// TIA Portal V15.1 export
// export: Created 2024-05-17T05:38:38.7642875Z, ExportSetting WithDefaults, DisplayName Totally Integrated Automation Portal, DisplayVersion V15.1 Update 5, DisplayName TIA Portal Openness, DisplayVersion V15.1 Update 5, DisplayName SINAMICS Startdrive Advanced, DisplayVersion V15.1, DisplayName G130, G150, S120, S150, SINAMICS MV, S210, DisplayVersion V15.1, DisplayName G110M, G120, G120C, G120D, G120P, DisplayVersion V15.1, DisplayName STEP 7 Professional, DisplayVersion V15.1 Update 5, DisplayName STEP 7 Safety, DisplayVersion V15.1, DisplayName WinCC Professional, DisplayVersion V15.1 Update 5, DisplayName SIMATIC Visualization Architect, DisplayVersion V15.1
FUNCTION_BLOCK "LGBAndonHCall"   // FB6687, FBD
TITLE = LGBAndonHCall
{ S7_Optimized_Access := 'TRUE' }
VERSION : 0.1
// This module will evaluate if an Andon HCall from pullcords and/or buttons is 
// valid and make the Hcall(AndonLight) active. It sends the result to LAndonxMConfig
// stored: AutoNumber false, IsIECCheckEnabled false, IsRetainMemResEnabled false, MemoryReserve 100, SetENOAutomatically False, UDAEnableTagReadback false
   VAR_INPUT
      I_HCall { ExternalAccessible := 'False'; ExternalVisible := 'False'; ExternalWritable := 'False'} : Bool;   // Input of the Human Call
      I_PartPresent { ExternalAccessible := 'False'; ExternalVisible := 'False'; ExternalWritable := 'False'} : Bool;   // Part is present on workstation
      C_HCallNumber { ExternalAccessible := 'False'; ExternalVisible := 'False'; ExternalWritable := 'False'} : Int;   // Address of the human call 1-32
      C_WorkStationNumber { ExternalAccessible := 'False'; ExternalVisible := 'False'; ExternalWritable := 'False'} : Int;   // Addeess of the Andon Station
   END_VAR
   VAR_OUTPUT
      O_AndonActiveSignal { ExternalAccessible := 'False'; ExternalVisible := 'False'; ExternalWritable := 'False'} : Bool;   // Output of the Hcall Light
      O_AndonCycleStpAfter { ExternalAccessible := 'False'; ExternalVisible := 'False'; ExternalWritable := 'False'} : Bool;   // Stop after end of cycle
   END_VAR
   VAR_IN_OUT
      IO_AndonDataExchange : "AndonDataExchangeVCG";   // Andon dataExchange
      H_HMI : "H_HMI";   // Animation
      H_GBAndonHCal : "H_GBAndonHCall";   // Animation
   END_VAR
   VAR RETAIN
      AndonActiveSignal { ExternalAccessible := 'False'; ExternalVisible := 'False'; ExternalWritable := 'False'} : Bool;
   END_VAR
   VAR
      AndonHCallDW { ExternalAccessible := 'False'; ExternalVisible := 'False'; ExternalWritable := 'False'} : DWord;
   END_VAR
   VAR RETAIN
      AndonHCallActiveBits { ExternalAccessible := 'False'; ExternalVisible := 'False'; ExternalWritable := 'False'} : Array[0..31] of Bool;
   END_VAR
   VAR
      LToggle_AndonHCall { ExternalAccessible := 'False'; ExternalVisible := 'False'; ExternalWritable := 'False'} : "LToggle";
      AndonHCallActive { ExternalAccessible := 'False'; ExternalVisible := 'False'; ExternalWritable := 'False'} : DWord;
      CorrectedHCallNumber { ExternalAccessible := 'False'; ExternalVisible := 'False'; ExternalWritable := 'False'} : Int;
   END_VAR
BEGIN

REGION Network 1: **** 1 - Inputs **** Get Andon HCall Active and copy it to a loacal variable
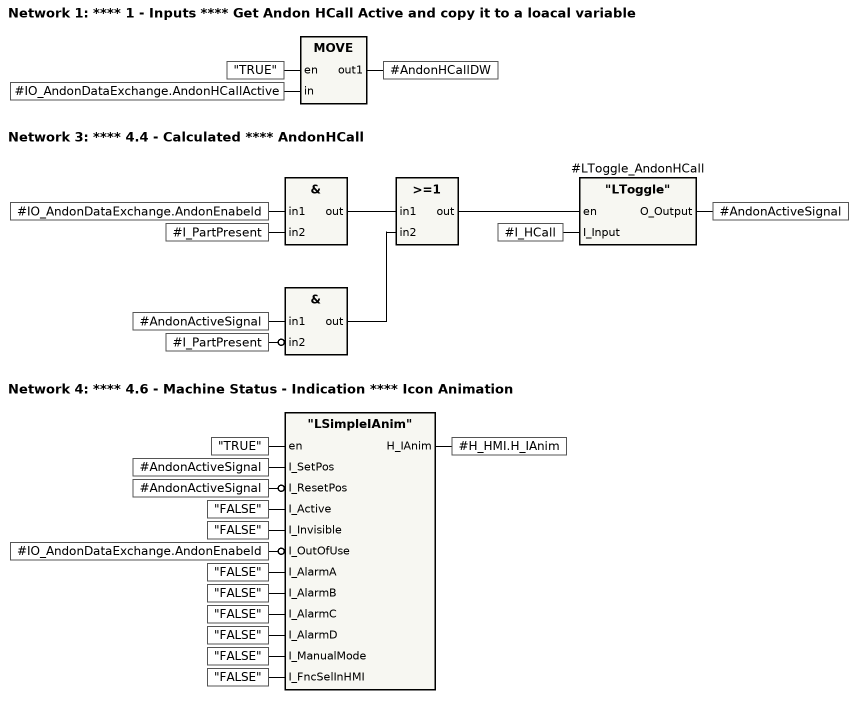
   IF "TRUE" THEN #AndonHCallDW := #IO_AndonDataExchange.AndonHCallActive; END_IF;
END_REGION

NETWORK
TITLE = **** 4.4 - Calculated **** Correct bit position in word -> HCall number
      L     #C_HCallNumber;
      L     1;
      -I;
      T     #CorrectedHCallNumber;

REGION Network 3: **** 4.4 - Calculated **** AndonHCall
   // * Andon must be enabeld
   // * Body musdt be in position
   // * Then toggle AndonCallStatus
   IF (#IO_AndonDataExchange.AndonEnabeld AND #I_PartPresent) OR (#AndonActiveSignal AND NOT #I_PartPresent) THEN
       #LToggle_AndonHCall(I_Input := #I_HCall, O_Output => #AndonActiveSignal);   // "LToggle"
   END_IF;
END_REGION

REGION Network 4: **** 4.6 - Machine Status - Indication **** Icon Animation
   IF "TRUE" THEN
       "LSimpleIAnim"(I_SetPos := #AndonActiveSignal,
                      I_ResetPos := NOT #AndonActiveSignal,
                      I_Active := "FALSE",
                      I_Invisible := "FALSE",
                      I_OutOfUse := NOT #IO_AndonDataExchange.AndonEnabeld,
                      I_AlarmA := "FALSE",
                      I_AlarmB := "FALSE",
                      I_AlarmC := "FALSE",
                      I_AlarmD := "FALSE",
                      I_ManualMode := "FALSE",
                      I_FncSelInHMI := "FALSE",
                      H_IAnim => #H_HMI.H_IAnim);
   END_IF;
END_REGION

REGION Network 5: **** 4.6 - Machine status - Indications **** Animation
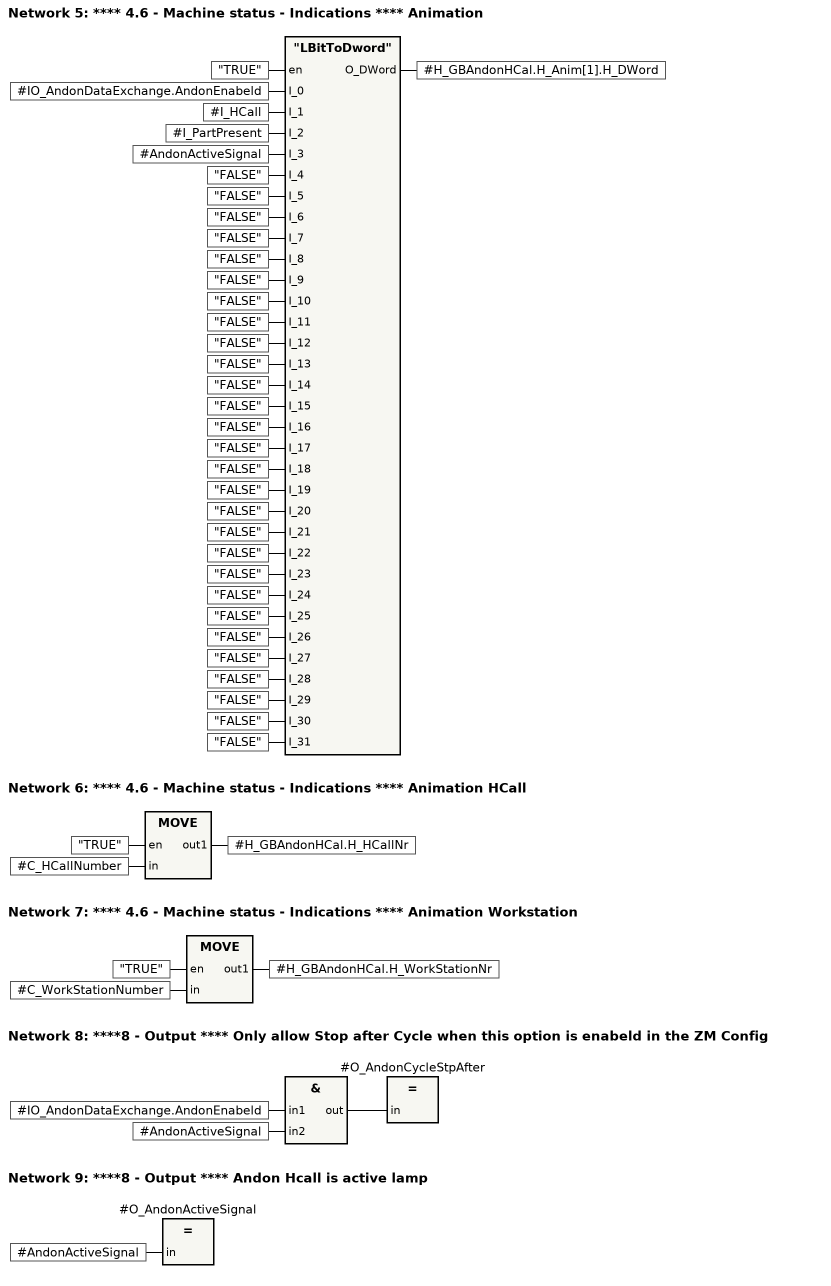
   IF "TRUE" THEN
       "LBitToDword"(I_0 := #IO_AndonDataExchange.AndonEnabeld,
                     I_1 := #I_HCall,
                     I_2 := #I_PartPresent,
                     I_3 := #AndonActiveSignal,
                     I_4 := "FALSE",
                     I_5 := "FALSE",
                     I_6 := "FALSE",
                     I_7 := "FALSE",
                     I_8 := "FALSE",
                     I_9 := "FALSE",
                     I_10 := "FALSE",
                     I_11 := "FALSE",
                     I_12 := "FALSE",
                     I_13 := "FALSE",
                     I_14 := "FALSE",
                     I_15 := "FALSE",
                     I_16 := "FALSE",
                     I_17 := "FALSE",
                     I_18 := "FALSE",
                     I_19 := "FALSE",
                     I_20 := "FALSE",
                     I_21 := "FALSE",
                     I_22 := "FALSE",
                     I_23 := "FALSE",
                     I_24 := "FALSE",
                     I_25 := "FALSE",
                     I_26 := "FALSE",
                     I_27 := "FALSE",
                     I_28 := "FALSE",
                     I_29 := "FALSE",
                     I_30 := "FALSE",
                     I_31 := "FALSE",
                     O_DWord => #H_GBAndonHCal.H_Anim[1].H_DWord);
   END_IF;
END_REGION

REGION Network 6: **** 4.6 - Machine status - Indications **** Animation HCall
   IF "TRUE" THEN #H_GBAndonHCal.H_HCallNr := #C_HCallNumber; END_IF;
END_REGION

REGION Network 7: **** 4.6 - Machine status - Indications **** Animation Workstation
   IF "TRUE" THEN #H_GBAndonHCal.H_WorkStationNr := #C_WorkStationNumber; END_IF;
END_REGION

REGION Network 8: ****8 - Output **** Only allow Stop after Cycle when this option is enabeld in the ZM Config
   #O_AndonCycleStpAfter := #IO_AndonDataExchange.AndonEnabeld AND #AndonActiveSignal;
END_REGION

REGION Network 9: ****8 - Output **** Andon Hcall is active lamp
   #O_AndonActiveSignal := #AndonActiveSignal;
END_REGION

NETWORK
TITLE = ****8 - Output **** Set corresponding bit in word
      A     #AndonActiveSignal;
      =     #AndonHCallActiveBits[#CorrectedHCallNumber];


REGION Network 11: ****8 - Output **** Set corresponding bit in word
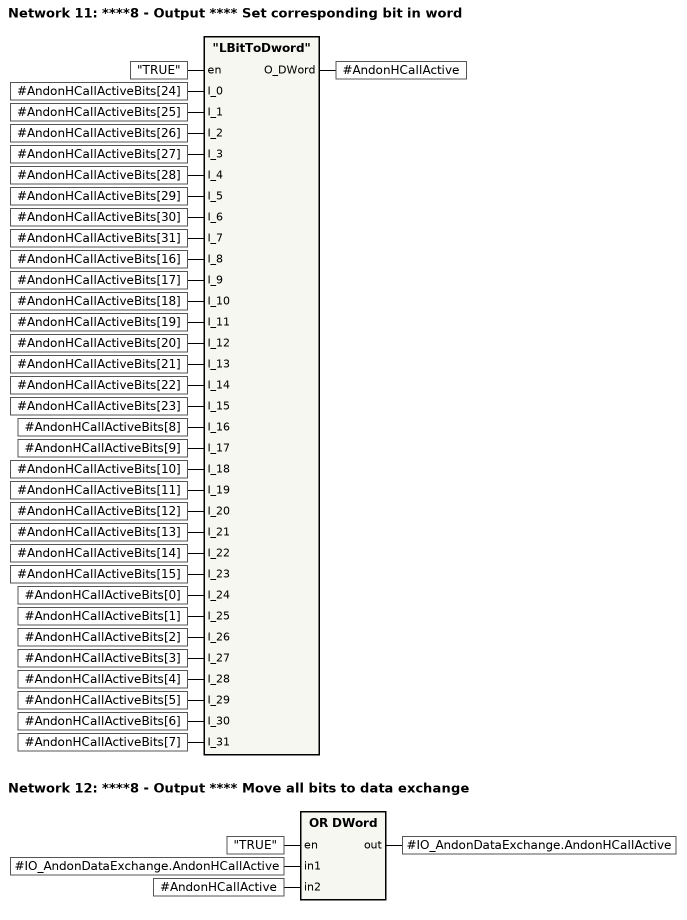
   IF "TRUE" THEN
       "LBitToDword"(I_0 := #AndonHCallActiveBits[24],
                     I_1 := #AndonHCallActiveBits[25],
                     I_2 := #AndonHCallActiveBits[26],
                     I_3 := #AndonHCallActiveBits[27],
                     I_4 := #AndonHCallActiveBits[28],
                     I_5 := #AndonHCallActiveBits[29],
                     I_6 := #AndonHCallActiveBits[30],
                     I_7 := #AndonHCallActiveBits[31],
                     I_8 := #AndonHCallActiveBits[16],
                     I_9 := #AndonHCallActiveBits[17],
                     I_10 := #AndonHCallActiveBits[18],
                     I_11 := #AndonHCallActiveBits[19],
                     I_12 := #AndonHCallActiveBits[20],
                     I_13 := #AndonHCallActiveBits[21],
                     I_14 := #AndonHCallActiveBits[22],
                     I_15 := #AndonHCallActiveBits[23],
                     I_16 := #AndonHCallActiveBits[8],
                     I_17 := #AndonHCallActiveBits[9],
                     I_18 := #AndonHCallActiveBits[10],
                     I_19 := #AndonHCallActiveBits[11],
                     I_20 := #AndonHCallActiveBits[12],
                     I_21 := #AndonHCallActiveBits[13],
                     I_22 := #AndonHCallActiveBits[14],
                     I_23 := #AndonHCallActiveBits[15],
                     I_24 := #AndonHCallActiveBits[0],
                     I_25 := #AndonHCallActiveBits[1],
                     I_26 := #AndonHCallActiveBits[2],
                     I_27 := #AndonHCallActiveBits[3],
                     I_28 := #AndonHCallActiveBits[4],
                     I_29 := #AndonHCallActiveBits[5],
                     I_30 := #AndonHCallActiveBits[6],
                     I_31 := #AndonHCallActiveBits[7],
                     O_DWord => #AndonHCallActive);
   END_IF;
END_REGION

REGION Network 12: ****8 - Output **** Move all bits to data exchange
   IF "TRUE" THEN
       #IO_AndonDataExchange.AndonHCallActive := #IO_AndonDataExchange.AndonHCallActive OR #AndonHCallActive;
   END_IF;
END_REGION
END_FUNCTION_BLOCK
